# EPICS substitutions: depo-orig/depoApp/Db/BK_1787B.substitutions
file TE_TC.template { pattern
{ Sys	, Dev		,PORT		, Chan	}
{ Depo	, "{PS:1}"	, Depo_PS1	, 1	}
}
